(* IEC 61131-3 sources: plc-vscode/tests/st/all/trust-platform/conformance/cases/edges/cfm_edges_r_f_trig_sequence_001, 1 file *)

(* ---- program.st ---- *)
PROGRAM Main
VAR
    r : R_TRIG;
    f : F_TRIG;
    clk : BOOL;
    q_r : BOOL;
    q_f : BOOL;
END_VAR

r(CLK := clk, Q => q_r);
f(CLK := clk, Q => q_f);
END_PROGRAM
